VAR_GLOBAL
	
	mb_Preactor:	LREAL	:= 0.0;
	mb_Treactor:	LREAL	:= 0.0;

END_VAR

(* stored: Version 1.1.0.1, ProductVersion 3.1.0.36
   GVL GVL_Modbus: Id {e76de713-a008-427e-b2ea-985e751f6dc8} *)
